FUNCTION_BLOCK CYCLE_DONE
  {SET_ATTRIBUTE(OpcUa, SERVICE)}
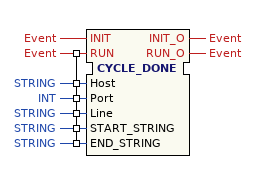
  EVENT_INPUT
    INIT;
    RUN WITH Host, Port, Line, START_STRING, END_STRING; {SET_ATTRIBUTE(OpcUa, Method)}
  END_EVENT
  EVENT_OUTPUT
    INIT_O;
    RUN_O;
  END_EVENT
  VAR_INPUT
    Host : STRING; {SET_ATTRIBUTE(OpcUa, Variable.RUN)}
    Port : INT; {SET_ATTRIBUTE(OpcUa, Variable.RUN)}
    Line : STRING; {SET_ATTRIBUTE(OpcUa, Variable.RUN)}
    START_STRING : STRING; {SET_ATTRIBUTE(OpcUa, Variable.RUN)}
    END_STRING : STRING; {SET_ATTRIBUTE(OpcUa, Variable.RUN)}
  END_VAR
END_FUNCTION_BLOCK
